Universal Robots PolyScope program: Main Program Left noweld.urp

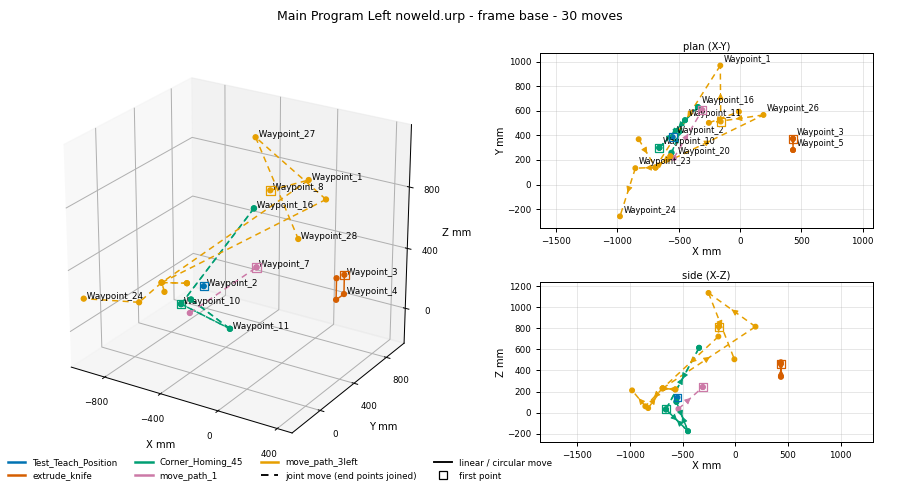
[picture p0: tool path of Main Program Left noweld.urp in frame base, 30 of 65 moves have a stored position in this frame; points joined in program order, loops and branches not executed]
Program Main Program Left noweld (installation=default directory=/programs createdIn=5.14.5 lastSavedIn=5.14.5 robotSerialNumber=20236801216)
Calibrated DH parameters: a=[-0.000021, -0.748897, -0.28186, -0.00004, -0.000055, 0]; d=[0.236225, -424.082933, -1564.66872, 1988.95162, 0.159094, 0.153873]; alpha=[1.570844, 0.001002, 0.000337, 1.571488, -1.569996, 0]; deltaTheta=[0, -0.516316, 5.626292, 1.173211, 0.000001, 0]
InitVariablesNode variables(variable(name=freedrive_m_var, expression=False))
Robot Program (runOnlyOnce=true)
  'start of main program'
  SafeHome (positionOptionType=SPEED_AND_ACCELERATION speed=1.047198 acceleration=1.396263 nextMotionTime=2)
  Set NoAction tcp=pretend_w_top
  Script: Test_Teach_Position()
  Set NoAction tcp=pretend_w_top
  Script: Corner_Homing_45()
  Set NoAction tcp=pretend_welder
  Script: extrude_knife()
  Script file /programs/analyze_touchpoints.script
    | # this file creates the function for analyzing touchpoints
    | # define pi
    | pi = 3.1415926535
    | 
    | # this is the main entry point for calculations.
    | # it takes in the 5 points, analyzes the shape of the box, and then calculates path points and returns them
    | # specifically for Down, Over, then Around (DOtA)
    | # specifically for right-sided boxes (vertical weld on right side of edge)
    | def main_calculate_right(p11, p12, p21, p22, p3, p13, p23):
    |     struct1 = analyze_touchpoints_only(p11, p12, p21, p22, p3)
    |     list1 = analyze_vertical_touchpoints(p11, p12, p13, p21, p22, p23, p3)
    |     struct2 = calculate_DOtA_points_right(struct1, list1)
    |     return struct2
    | end
    | 
    | # this is the main entry point for calculations.
    | # it takes in the 5 points, analyzes the shape of the box, and then calculates path points and returns them
    | # specifically for Down, Over, then Around (DOtA)
    | # specifically for left-sided boxes (vertical weld on left side of edge)
    | def main_calculate_left(p11, p12, p21, p22, p3):
    |     struct1 = analyze_touchpoints_only(p11, p12, p21, p22, p3)
    |     struct2 = calculate_DOtA_points_left(struct1)
    |     return struct2
    | end
    | 
    | # it takes 5 arguments as points
    | # it returns a struct containing: (pointintersect, pointapproach1, pointapproach2, point1, point2, point3, point4, point5, pointreturn1, heading1, heading2, heading3, path2r1, path2r2, path2l1, path2l2)
    | # specifically for Around then Up (AtU)
    | def analyze_touchpoints(p11, p12, p21, p22, p3):
    |   # FIND THE INTERSECTION
    |   # comment get the z
    |   zcoord=p3[2]
    | 
    |   # get the raw points from the first line
    |   l1p1x=p11[0]
    |   l1p1y=p11[1]
    |   l1p2x=p12[0]
    |   l1p2y=p12[1]
    | 
    |   # equate the first line in 2d space
    |   ml1 = (l1p2y-l1p1y) / (l1p2x-l1p1x)
    | 
    |   # b = y - mx
    |   bl1 = l1p1y - ml1 * l1p1x
    | 
    |   # get the raw points from the second line
    |   l2p1x=p21[0]
    |   l2p1y=p21[1]
    |   l2p2x=p22[0]
    |   l2p2y=p22[1]
    | 
    |   # equate the second line in 2d space
    |   ml2 = (l2p2y-l2p1y) / (l2p2x-l2p1x)
    | 
    |   # b = y - mx
    |   bl2 = l2p1y - ml2 * l2p1x
    | 
    | 
    |   # find the intersection of the two lines
    |   # m1x+b1 = m2x+b2
    |   # m1x - m2x = b2 - b1
    |   # x = (b2-b1) / (m1-m2)
    |   xintersect = (bl2-bl1) / (ml1-ml2)
    |   yintersect = ml1 * xintersect + bl1
    | 
    |   #FIND THE VECTORS
    |   #define a vector from the intersection to the second point on the first line
    |   l1delxfull = l1p2x - xintersect
    |   l1delyfull = l1p2y - yintersect
    | 
    |   l1delmag = sqrt(l1delxfull*l1delxfull + l1delyfull*l1delyfull)
    | 
    |   l1delxunit = l1delxfull / l1delmag
    |   l1delyunit = l1delyfull / l1delmag
    | 
    |   #define a vector from the intersection to the second point on the second line
    |   l2delxfull = l2p2x - xintersect
    |   l2delyfull = l2p2y - yintersect
    | 
    |   l2delmag = sqrt(l2delxfull*l2delxfull + l2delyfull*l2delyfull)
    | 
    |   l2delxunit = l2delxfull / l2delmag
    |   l2delyunit = l2delyfull / l2delmag
    | 
    |   # FIND THE FOUR POINTS ON THE LINES
    |   # find locations 8 inches away from  intersect point
    |   # CONST
    |   welddistance = 8
    |   roundoverdistance = 0.05
    |   zup = .375
    |   # inches
    |   wd = welddistance * 25.4 / 1000
    |   rod = roundoverdistance * 25.4 / 1000
    |   zup = zup * 25.4 / 1000
    | 
    |   # now we have the unit vector. extend the weld distance from the intersection
    |   x = xintersect + l1delxunit * wd
    |   y = yintersect + l1delyunit * wd
    |   z = zcoord + zup
    | 
    |   point1 = p[x,y,z,1.570796,0,0] # dummy orientation for now
    | 
    |   x = xintersect + l1delxunit * rod
    |   y = yintersect + l1delyunit * rod
    | 
    |   point2 = p[x,y,z,1.570796,0,0]
    | 
    |   # now we have the unit vector. extend the weld distance from the intersection
    |   x = xintersect + l2delxunit * wd
    |   y = yintersect + l2delyunit * wd
    | 
    |   point5 = p[x,y,z,0,-1.570796,0]
    | 
    |   x = xintersect + l2delxunit * rod
    |   y = yintersect + l2delyunit * rod
    | 
    |   point4 = p[x,y,z,0,-1.570796,0]
    | 
    |   #DEFINE APPROACH POINTS
    |   pointintersect = p[xintersect,yintersect,zcoord,0,0,0]
    |   pointapproach1 = p[xintersect+0.1,yintersect+0.1,z,1.570796,0,0]
    |   pointapproach2 = p[point1[0], point1[1]+0.1, point1[2], point1[3], point1[4], point1[5]]
    |   pointreturn1 = p[point5[0]+0.1, point5[1], point5[2], point5[3], point5[4], point5[5]]
    | 
    |   #FIND HEADINGS
    |   #for each heading, find the angle of the line with respect to the pos x axis. then add/subtract 90 degrees because you want to be perpendicular to that
    |   headingvector1 = convert_uv_to_heading(l1delxunit, l1delyunit)
    |   headingvector2 = convert_uv_to_heading(l2delxunit, l2delyunit)
    |   # find halfway heading
    |   heading2 = (headingvector1 + headingvector2)/2
    |   # find headings that the robot should face while traveling, perpendicular to the vectors of the sides of the box
    |   heading1 = headingvector1 + pi/2
    |   heading3 = headingvector2 - pi/2
    | 
    |   #FIND POINT 3
    |   #see if we have to / can find point 3
    |   findpoint3 = True
    |   if roundoverdistance == 0:
    |     findpoint3 = False
    |   end
    |   if findpoint3:
    |     # i need to find the point3 such that the arc from p2 to p3 to p4 is tangent to p1-p2 and p4-p5. making this a smooth path will be good
    |     # the direction of movement is from pointintersect in the direction of heading2
    |     # how much movement though? this will depend on whether it is actually a 90 degree angle or not.
    |     # first, find the perpendicular lines through points 2 and 4
    |     perp2 = find_perpendicular_line(ml1, point2[0], point2[1])
    |     perp4 = find_perpendicular_line(ml2, point4[0], point4[1])
    |     # next, find the intersection of those two lines
    |     perpintersect = find_intersection(perp2[0], perp2[1], perp4[0], perp4[1])
    |     radiusofcircle = distance_between(perpintersect[0], perpintersect[1], 0, point2[0], point2[1], 0)
    |     # find a vector the direction of heading2
    |     uvx = cos(heading2)
    |     uvy = sin(heading2)
    |     # compute point3. pass in negative radius because the direction is into the tank but we want to move from the intersection out to the rounded edge.
    |     point3coords = add_vectordistance_to_point(perpintersect[0], perpintersect[1], z, uvx, uvy, 0, -1 * radiusofcircle)
    |     point3 = p[point3coords[0], point3coords[1], point3coords[2], 0, 0, 0]
    |   end
    | 
    |   #APPLY ACTUAL RXRYRZ TO POINTS
    |   # convert the headings to rxryrz and insert those values into the relevant points
    |   rxryrz = convert_heading_to_axang(heading1)
    |   rx = rxryrz[0]
    |   ry = rxryrz[1]
    |   rz = rxryrz[2]
    |   pointapproach1 = p[pointapproach1[0], pointapproach1[1], pointapproach1[2], rx, ry, rz]
    |   pointapproach2 = p[pointapproach2[0], pointapproach2[1], pointapproach2[2], rx, ry, rz]
    |   point1 = p[point1[0], point1[1], point1[2], rx, ry, rz]
    |   point2 = p[point2[0], point2[1], point2[2], rx, ry, rz]
    |   rxryrz = convert_heading_to_axang(heading2)
    |   rx = rxryrz[0]
    |   ry = rxryrz[1]
    |   rz = rxryrz[2]
    |   if findpoint3:
    |     point3 = p[point3[0], point3[1], point3[2], rx, ry, rz]
    |   else:
    |     point3 = point2
    |   end
    |   rxryrz = convert_heading_to_axang(heading3)
    |   rx = rxryrz[0]
    |   ry = rxryrz[1]
    |   rz = rxryrz[2]
    |   point4 = p[point4[0], point4[1], point4[2], rx, ry, rz]
    |   point5 = p[point5[0], point5[1], point5[2], rx, ry, rz]
    |   pointreturn1 = p[pointreturn1[0], pointreturn1[1], pointreturn1[2], rx, ry, rz]
    | 
    |   #find path2 (the part that goes up)
    |   four_vertical_points = find_vertical_points(pointintersect, l1delxunit, l1delyunit, l2delxunit, l2delyunit, zup, wd, heading1, heading3)
    |   path2r1 = four_vertical_points[0]
    |   path2r2 = four_vertical_points[1]
    |   path2l1 = four_vertical_points[2]
    |   path2l2 = four_vertical_points[3]
    | 
    |   #RETURN STRUCT
    |   ret = struct(pointintersect=pointintersect, pointapproach1=pointapproach1, pointapproach2=pointapproach2, point1=point1, point2=point2, point3=point3, point4=point4, point5=point5, pointreturn1=pointreturn1, heading1=heading1, heading2=heading2, heading3=heading3, path2r1=path2r1, path2r2=path2r2, path2l1=path2l1, path2l2=path2l2)
    |   return ret
    | end
    | 
    | # it takes 5 arguments as points
    | # it returns a struct containing: (pointintersect, heading1, heading2, heading3, l1delxunit, l1delyunit, l2delxunit, l2delyunit)
    | def analyze_touchpoints_only(p11, p12, p21, p22, p3):
    |   # FIND THE INTERSECTION
    |   # comment get the z
    |   zcoord=p3[2]
    | 
    |   # get the raw points from the first line
    |   l1p1x=p11[0]
    |   l1p1y=p11[1]
    |   l1p2x=p12[0]
    |   l1p2y=p12[1]
    | 
    |   # equate the first line in 2d space
    |   ml1 = (l1p2y-l1p1y) / (l1p2x-l1p1x)
    | 
    |   # b = y - mx
    |   bl1 = l1p1y - ml1 * l1p1x
    | 
    |   # get the raw points from the second line
    |   l2p1x=p21[0]
    |   l2p1y=p21[1]
    |   l2p2x=p22[0]
    |   l2p2y=p22[1]
    | 
    |   # equate the second line in 2d space
    |   ml2 = (l2p2y-l2p1y) / (l2p2x-l2p1x)
    | 
    |   # b = y - mx
    |   bl2 = l2p1y - ml2 * l2p1x
    | 
    | 
    |   # find the intersection of the two lines
    |   # m1x+b1 = m2x+b2
    |   # m1x - m2x = b2 - b1
    |   # x = (b2-b1) / (m1-m2)
    |   xintersect = (bl2-bl1) / (ml1-ml2)
    |   yintersect = ml1 * xintersect + bl1
    | 
    |   pointintersect = p[xintersect,yintersect,zcoord,0,0,0]
    | 
    |   #FIND THE VECTORS
    |   #define a vector from the intersection to the second point on the first line
    |   l1delxfull = l1p2x - xintersect
    |   l1delyfull = l1p2y - yintersect
    | 
    |   l1delmag = sqrt(l1delxfull*l1delxfull + l1delyfull*l1delyfull)
    | 
    |   l1delxunit = l1delxfull / l1delmag
    |   l1delyunit = l1delyfull / l1delmag
    | 
    |   #define a vector from the intersection to the second point on the second line
    |   l2delxfull = l2p2x - xintersect
    |   l2delyfull = l2p2y - yintersect
    | 
    |   l2delmag = sqrt(l2delxfull*l2delxfull + l2delyfull*l2delyfull)
    | 
    |   l2delxunit = l2delxfull / l2delmag
    |   l2delyunit = l2delyfull / l2delmag
    | 
    |   #FIND HEADINGS
    |   #for each heading, find the angle of the line with respect to the pos x axis. then add/subtract 90 degrees because you want to be perpendicular to that
    |   headingvector1 = convert_uv_to_heading(l1delxunit, l1delyunit)
    |   headingvector2 = convert_uv_to_heading(l2delxunit, l2delyunit)
    |   # find halfway heading
    |   heading2 = (headingvector1 + headingvector2)/2
    |   # find headings that the robot should face while traveling, perpendicular to the vectors of the sides of the box
    |   heading1 = headingvector1 + pi/2
    |   heading3 = headingvector2 - pi/2
    | 
    |   #RETURN STRUCT
    |   ret = struct(pointintersect=pointintersect, heading1=heading1, heading2=heading2, heading3=heading3, l1delxunit=l1delxunit, l1delyunit=l1delyunit, l2delxunit=l2delxunit, l2delyunit=l2delyunit)
    |   return ret
    | end
    | 
    | # given a struct from analyze_touchpoints_only(), calculate the points
    | def calculate_DOtA_points_right(struct1, listleans):
    |     # get the stuff from the struct
    |     pointintersect = struct1[0]
    |     heading1 = struct1[1]
    |     heading2 = struct1[2]
    |     heading3 = struct1[3]
    |     l1delxunit = struct1[4]
    |     l1delyunit = struct1[5]
    |     l2delxunit = struct1[6]
    |     l2delyunit = struct1[7]
    | 
    |     # FIND THE POINTS ON THE LINES OF THE FIRST TURN PATH
    |     # find locations 8 inches away from  intersect point
    |     # CONST
    |     welddistance1 = 8 # vertical weld distance
    |     welddistance2 = 6 # first path second leg
    |     welddistance3 = 8 # second path second leg
    |     zup = .375
    |     # inches
    |     wd1 = welddistance1 * 25.4 / 1000
    |     wd2 = welddistance2 * 25.4 / 1000
    |     wd3 = welddistance3 * 25.4 / 1000
    |     zup = zup * 25.4 / 1000
    | 
    |     x = pointintersect[0] + l1delxunit * zup
    |     y = pointintersect[1] + l1delyunit * zup
    |     z = pointintersect[2] + zup
    | 
    |     #apply actual rxryrz to points
    |     # convert the headings to rxryrz and insert those values into the relevant points
    |     rxryrz = convert_heading_to_axang_preheatdown(heading1)
    |     rx = rxryrz[0]
    |     ry = rxryrz[1]
    |     rz = rxryrz[2]
    | 
    |     point1 = p[x + wd1*listleans[0], y + wd1*listleans[1], z + wd1, rx, ry, rz] # add in the listleans factor to follow the face of the box as we move up
    |     point2 = p[x, y, z, rx, ry, rz]
    | 
    |     # convert the headings to rxryrz and insert those values into the relevant points
    |     rxryrz = convert_heading_to_axang_ccw(heading1)
    |     rx = rxryrz[0]
    |     ry = rxryrz[1]
    |     rz = rxryrz[2]
    | 
    |     point4 = p[x, y, z, rx, ry, rz]
    |     x = x + l1delxunit * wd2
    |     y = y + l1delyunit * wd2
    |     point5 = p[x, y, z, rx, ry, rz]
    | 
    |     # FIND THE POINTS ON THE LINES OF THE SECOND AROUND PATH
    |     roundoverdistance = 0.05
    |     rod = roundoverdistance * 25.4 / 1000
    | 
    |     # now we have the unit vector. extend the weld distance from the intersection
    |     x = pointintersect[0] + l1delxunit * (zup)
    |     y = pointintersect[1] + l1delyunit * zup
    |     # convert the headings to rxryrz and insert those values into the relevant points
    |     rxryrz = convert_heading_to_axang(heading1)
    |     rx = rxryrz[0]
    |     ry = rxryrz[1]
    |     rz = rxryrz[2]
    |     point_1 = p[x, y, z, rx, ry, rz]
    | 
    |     x = pointintersect[0] + l1delxunit * rod
    |     y = pointintersect[1] + l1delyunit * rod
    |     point_2 = p[x, y, z, rx, ry, rz]
    | 
    |     # now we have the unit vector. extend the weld distance from the intersection
    |     x = pointintersect[0] + l2delxunit * wd3
    |     y = pointintersect[1] + l2delyunit * wd3
    |     # convert the headings to rxryrz and insert those values into the relevant points
    |     rxryrz = convert_heading_to_axang(heading3)
    |     rx = rxryrz[0]
    |     ry = rxryrz[1]
    |     rz = rxryrz[2]
    |     point_5 = p[x, y, z, rx, ry, rz]
    | 
    |     x = pointintersect[0] + l2delxunit * rod
    |     y = pointintersect[1] + l2delyunit * rod
    |     point_4 = p[x, y, z, rx, ry, rz]
    | 
    |     #FIND POINT 3
    |     # by calling analyze_touchpoints()
    |     atret = analyze_touchpoints(point_2, point_1, point_4, point_5, pointintersect)
    |     point_3 = atret[5]
    | 
    | 
    |     struct2 = struct(point1=point1, point2=point2, point4=point4, point5=point5, point_1=point_1, point_2=point_2, point_3=point_3, point_4=point_4, point_5=point_5)
    |     return struct2
    | end
    | 
    | # given a struct from analyze_touchpoints_only(), calculate the points
    | def calculate_DOtA_points_left(struct1):
    |     # get the stuff from the struct
    |     pointintersect = struct1[0]
    |     heading1 = struct1[1]
    |     heading2 = struct1[2]
    |     heading3 = struct1[3]
    |     l1delxunit = struct1[4]
    |     l1delyunit = struct1[5]
    |     l2delxunit = struct1[6]
    |     l2delyunit = struct1[7]
    | 
    |     # FIND THE POINTS ON THE LINES OF THE FIRST TURN PATH
    |     # find locations 8 inches away from  intersect point
    |     # CONST
    |     welddistance = 8
    |     zup = .375
    |     # inches
    |     wd = welddistance * 25.4 / 1000
    |     zup = zup * 25.4 / 1000
    | 
    |     x = pointintersect[0] + l2delxunit * zup
    |     y = pointintersect[1] + l2delyunit * zup
    |     z = pointintersect[2] + zup
    | 
    |     #apply actual rxryrz to points
    |     # convert the headings to rxryrz and insert those values into the relevant points
    |     rxryrz = convert_heading_to_axang_preheatdown(heading3)
    |     rx = rxryrz[0]
    |     ry = rxryrz[1]
    |     rz = rxryrz[2]
    | 
    |     point1 = p[x, y, z + wd, rx, ry, rz]
    |     point2 = p[x, y, z, rx, ry, rz]
    | 
    |     # convert the headings to rxryrz and insert those values into the relevant points
    |     rxryrz = convert_heading_to_axang(heading3)
    |     rx = rxryrz[0]
    |     ry = rxryrz[1]
    |     rz = rxryrz[2]
    | 
    |     point4 = p[x, y, z, rx, ry, rz]
    |     x = x + l2delxunit * wd
    |     y = y + l2delyunit * wd
    |     point5 = p[x, y, z, rx, ry, rz]
    | 
    |     # FIND THE POINTS ON THE LINES OF THE SECOND AROUND PATH
    |     roundoverdistance = 0.05
    |     rod = roundoverdistance * 25.4 / 1000
    | 
    |     # now we have the unit vector. extend the weld distance from the intersection
    |     x = pointintersect[0] + l2delxunit * (zup)
    |     y = pointintersect[1] + l2delyunit * zup
    |     # convert the headings to rxryrz and insert those values into the relevant points
    |     rxryrz = convert_heading_to_axang_ccw(heading3)
    |     rx = rxryrz[0]
    |     ry = rxryrz[1]
    |     rz = rxryrz[2]
    |     point_1 = p[x, y, z, rx, ry, rz]
    | 
    |     x = pointintersect[0] + l2delxunit * rod
    |     y = pointintersect[1] + l2delyunit * rod
    |     point_2 = p[x, y, z, rx, ry, rz]
    | 
    |     # now we have the unit vector. extend the weld distance from the intersection
    |     x = pointintersect[0] + l1delxunit * wd
    |     y = pointintersect[1] + l1delyunit * wd
    |     # convert the headings to rxryrz and insert those values into the relevant points
    |     rxryrz = convert_heading_to_axang_ccw(heading1)
    |     rx = rxryrz[0]
    |     ry = rxryrz[1]
    |     rz = rxryrz[2]
    |     point_5 = p[x, y, z, rx, ry, rz]
    | 
    |     x = pointintersect[0] + l1delxunit * rod
    |     y = pointintersect[1] + l1delyunit * rod
    |     point_4 = p[x, y, z, rx, ry, rz]
    | 
    |     #FIND POINT 3
    |     # by calling analyze_touchpoints()
    |     atret = analyze_touchpoints(point_2, point_1, point_4, point_5, pointintersect)
    |     point_3 = atret[5]
    |     #point 3 will not have the correct rxryrz though because now the gun needs to be face up.
    |     rxryrz = convert_heading_to_axang_ccw(heading2)
    |     rx = rxryrz[0]
    |     ry = rxryrz[1]
    |     rz = rxryrz[2]
    |     point_3 = p[point_3[0], point_3[1], point_3[2], rx, ry, rz]
    | 
    |     struct2 = struct(point1=point1, point2=point2, point4=point4, point5=point5, point_1=point_1, point_2=point_2, point_3=point_3, point_4=point_4, point_5=point_5)
    |     return struct2
    | end
    | 
    | # this function analyzes the vertical points
    | # calculates the slope of the edge in question
    | # specifically, for each inch up in the z direction, what is the change in x and change in y direction
    | # returns a list of [nx, ny]
    | def analyze_vertical_touchpoints(p11, p12, p13, p21, p22, p23, p3):
    |     # first, find the equations of the planes from the 6 points
    |     plane1 = findplane(p11, p12, p13)
    |     plane2 = findplane(p21, p22, p23)
    |     # Find the Direction Vector of the Line: The direction vector d of the line of intersection can be found by taking the cross product of the normal vectors of each plane (a, b, and c)
    |     nx = plane1[1]*plane2[2] - plane1[2]*plane2[1]
    |     ny = plane1[2]*plane2[0] - plane1[0]*plane2[2]
    |     nz = plane1[0]*plane2[1] - plane1[1]*plane2[0]
    |     # normalize the vector so the z length is 1
    |     multiplier = 1 / nz
    |     nx = nx * multiplier
    |     ny = ny * multiplier
    |     nz = nz * multiplier # should become equal to 1
    |     ret = [nx, ny]
    |     return ret
    | end
    | 
    | # given 3 points, this finds the plane and its equation
    | # rereturns ax + by + cz + d = 0 in a list of [a, b, c, d]
    | def findplane(p11, p12, p13):
    |     # extract coordinates
    |     x1 = p11[0]
    |     y1 = p11[1]
    |     z1 = p11[2]
    |     x2 = p12[0]
    |     y2 = p12[1]
    |     z2 = p12[2]
    |     x3 = p13[0]
    |     y3 = p13[1]
    |     z3 = p13[2]
    |     # create vectors from the points
    |     v1x = x2-x1
    |     v1y = y2-y1
    |     v1z = z2-z1
    |     v2x = x3-x1
    |     v2y = y3-y1
    |     v2z = z3-z1
    |     #calculate the normal vector using the cross product
    |     nx = v1y*v2z - v1z*v2y # i component
    |     ny = v1z*v2x - v1x*v2z # j component
    |     nz = v1x*v2y - v1y*v2x # k component
    |     # calculate d in the plane equation
    |     d = -1 * (nx*x1 + ny*y1 + nz*z1)
    |     ret = [nx, ny, nz, d]
    |     return ret
    | end
    | 
    | # given a heading, (ccw from +x axis), find the mx+b slope
    | # fails if exactly vertical
    | def get_slope_from_heading(heading):
    |     return tan(heading)
    | end
    | 
    | 
    | 
    | # this function finds the points (and rxryrz) of the 2 points (start and end) of vertical weld section
    | def find_vertical_points(pointintersect, l1delxunit, l1delyunit, l2delxunit, l2delyunit, offset, wd, heading1, heading3):
    | 
    |   # find right side stuff
    |   # find the point in 3d space that is .375 up and .375 over
    |   x = pointintersect[0] + l1delxunit * offset
    |   y = pointintersect[1] + l1delyunit * offset
    |   z = pointintersect[2] + offset
    |   # find rxryrz
    |   rxryrz = convert_heading_to_axang_preheatup(heading1)
    |   rx = rxryrz[0]
    |   ry = rxryrz[1]
    |   rz = rxryrz[2]
    |   path2r1 = p[x, y, z, rx, ry, rz]
    |   path2r2 = p[x, y, z + wd, rx, ry, rz]
    | 
    |   # find left side
    |   # find the point in 3d space that is .375 up and .375 over
    |   x = pointintersect[0] + l2delxunit * offset
    |   y = pointintersect[1] + l2delyunit * offset
    |   z = pointintersect[2] + offset
    |   # find rxryrz
    |   rxryrz = convert_heading_to_axang_preheatup(heading3)
    |   rx = rxryrz[0]
    |   ry = rxryrz[1]
    |   rz = rxryrz[2]
    |   path2l1 = p[x, y, z, rx, ry, rz]
    |   path2l2 = p[x, y, z + wd, rx, ry, rz]
    | 
    |   ret = struct(path2r1=path2r1, path2r2=path2r2, path2l1=path2l1, path2l2=path2l2)
    |   return ret
    | end
    | 
    | # this function converts a unit vector to its heading angle ccw from x+ axis
    | # takes uvx and uvy
    | # returns heading in radians
    | def convert_uv_to_heading(uvx, uvy):
    |   baseang = atan(uvy/uvx)
    |   if uvx < 0:
    |     ang = baseang + pi
    |   elif uvy < 0:
    |     ang = baseang + pi * 2
    |   else:
    |     ang = baseang
    |   end
    |   return ang
    | end
    | 
    | # this function finds the equation of a line, perpendicular to a given line, and going through a given point
    | # takes 3 arguments: m (the original line's slope), x (point's x coord), y (point's y coord). the b of the original line is not needed
    | # returns a list of [m,b] (the slope and intercept of the new line)
    | def find_perpendicular_line(origm, x, y):
    |   m = (1/origm) * -1
    |   b = y - m*x
    |   ret = [m, b]
    |   return ret
    | end
    | 
    | # this function finds the intersection point between two lines in the xy plane
    | # takes 4 arguments: m1, b1, m2, b2
    | # returns a list of [x,y] (the point of intersection)
    | def find_intersection(m1, b1, m2, b2):
    |   # m1x+b1 = m2x+b2
    |   # m1x - m2x = b2 - b1
    |   # x = (b2-b1) / (m1-m2)
    |   x = (b2-b1) / (m1-m2)
    |   y = m1 * x + b1
    |   ret = [x, y]
    |   return ret
    | end
    | 
    | # this function finds the distance between 2 points in 3d space
    | # it takes 6 arguments: x1, y1, z1, x2, y2, z2
    | # it returns a distance
    | def distance_between(x1, y1, z1, x2, y2, z2):
    |   distsquared = (x2-x1)*(x2-x1)+(y2-y1)*(y2-y1)+(z2-z1)*(z2-z1)
    |   dist = sqrt(distsquared)
    |   return dist
    | end
    | 
    | # this function takes a point, a unit vector, and a distance, and adds the distance to the point in the direction of the unit vector (3d space)
    | # it returns a point as a list of coordinates
    | def add_vectordistance_to_point(xi, yi, zi, uvx, uvy, uvz, delta):
    |   xf = xi + uvx * delta
    |   yf = yi + uvy * delta
    |   zf = zi + uvz * delta
    |   ret = [xf, yf, zf]
    |   return ret
    | end
    | 
    | # this function converts a heading (ccw radians from the positive x axis) into rxryrz to be put into a point p[]
    | # this will point the gun in this heading with the bottom side of the gun facing up.
    | # the values used in this program were calculated by doing rotation matrix math in the file on WI-CALVINB10 C. Documents. Theory for converting rotations into axis angle representations
    | def convert_heading_to_axang(heading):
    |  axisxraw = -1 * sin(heading)
    |  axisyraw = cos(heading) + 1
    |  axiszraw = sin(heading)
    | 
    |  magnitude = sqrt(axisxraw*axisxraw + axisyraw*axisyraw + axiszraw*axiszraw)
    | 
    |  axisxunit = axisxraw / magnitude
    |  axisyunit = axisyraw / magnitude
    |  axiszunit = axiszraw / magnitude
    | 
    |  angle = acos( (cos(heading) - 1) / 2 )
    | 
    |  rxout = axisxunit * angle
    |  ryout = axisyunit * angle
    |  rzout = axiszunit * angle
    | 
    |  return [rxout, ryout, rzout]
    | end
    | 
    | # this function converts a heading (ccw radians from the positive x axis) into rxryrz to be put into a point p[]
    | # this will point the gun in this heading with the preheat side of the gun tip facing up. Used for welding in a vertical path.
    | # the values used in this program were calculated by doing rotation matrix math in the file on WI-CALVINB10 C. Documents. Theory for converting rotations into axis angle representations
    | def convert_heading_to_axang_preheatup(heading):
    |  axisxraw = -sin(heading) + 1
    |  axisyraw = cos(heading)
    |  axiszraw = cos(heading)
    | 
    |  magnitude = sqrt(axisxraw*axisxraw + axisyraw*axisyraw + axiszraw*axiszraw)
    | 
    |  axisxunit = axisxraw / magnitude
    |  axisyunit = axisyraw / magnitude
    |  axiszunit = axiszraw / magnitude
    | 
    |  angle = acos( (-sin(heading) - 1) / 2 )
    | 
    |  rxout = axisxunit * angle
    |  ryout = axisyunit * angle
    |  rzout = axiszunit * angle
    | 
    |  return [rxout, ryout, rzout]
    | end
    | 
    | # this function converts a heading (ccw radians from the positive x axis) into rxryrz to be put into a point p[]
    | # this will point the gun in this heading with the preheat side of the gun tip facing down. Used for welding in a vertical path downwards.
    | # the values used in this program were calculated by doing rotation matrix math in the file on WI-CALVINB10 C. Documents. Theory for converting rotations into axis angle representations
    | def convert_heading_to_axang_preheatdown(heading):
    |  axisxraw = -sin(heading) - 1
    |  axisyraw = cos(heading)
    |  axiszraw = -cos(heading)
    | 
    |  magnitude = sqrt(axisxraw*axisxraw + axisyraw*axisyraw + axiszraw*axiszraw)
    | 
    |  axisxunit = axisxraw / magnitude
    |  axisyunit = axisyraw / magnitude
    |  axiszunit = axiszraw / magnitude
    | 
    |  angle = acos( (sin(heading) - 1) / 2 )
    | 
    |  rxout = axisxunit * angle
    |  ryout = axisyunit * angle
    |  rzout = axiszunit * angle
    | 
    |  return [rxout, ryout, rzout]
    | end
    | 
    | # this function converts a heading (ccw radians from the positive x axis) into rxryrz to be put into a point p[]
    | # this will point the gun in this heading with the preheat side of the gun tip facing right. Used for welding counterclockwise around the box.
    | # the values used in this program were calculated by doing rotation matrix math in the file on WI-CALVINB10 C. Documents. Theory for converting rotations into axis angle representations
    | def convert_heading_to_axang_ccw(heading):
    |  axisxraw = -sin(heading)
    |  axisyraw = cos(heading) - 1
    |  axiszraw = -sin(heading)
    | 
    |  magnitude = sqrt(axisxraw*axisxraw + axisyraw*axisyraw + axiszraw*axiszraw)
    | 
    |  axisxunit = axisxraw / magnitude
    |  axisyunit = axisyraw / magnitude
    |  axiszunit = axiszraw / magnitude
    | 
    |  angle = acos( (-cos(heading) - 1) / 2 )
    | 
    |  rxout = axisxunit * angle
    |  ryout = axisyunit * angle
    |  rzout = axiszunit * angle
    | 
    |  return [rxout, ryout, rzout]
    | end
    | 
    | # this function is for getting the points along the path of the corner homing 45
    | # point0 is the point where they touched
    | def get_corner_homing_45_pathpoints(point0):
    |   p0x = point0[0]
    |   p0y = point0[1]
    |   p0z = point0[2]
    |   p0rx = point0[3]
    |   p0ry = point0[4]
    |   p0rz = point0[5]
    | 
    |   #constants
    |   #distances of how far away from point the touchpoints are
    |   d0 = 0.15 # how far from the box to retreat and approach
    |   d1 = 0.05 # first distance from init point
    |   d2 = 0.2 # second distance from init point
    |   d3 = 0.125 #vertical distance from first point
    |   sqrt2 = 0.707106781
    | 
    |   ph1 = p[p0x + d0, p0y, p0z + .05, p0rx, p0ry, p0rz] #approach point for turn
    | 
    |   ph2 = p[p0x+d0-d0*sqrt2-sqrt2*d1, p0y+d0*sqrt2+sqrt2*d1, p0z+.05, .445, -1.562, .483]
    |   ph3 = p[p0x+d0-d0*sqrt2-sqrt2*d2, p0y+d0*sqrt2+sqrt2*d2, p0z+.05, .445, -1.562, .483]
    |   ph4 = p[p0x+d0-d0*sqrt2-sqrt2*d1, p0y-d0*sqrt2-sqrt2*d1, p0z+.05, 1.699, 3.576, 1.841]
    |   ph5 = p[p0x+d0-d0*sqrt2-sqrt2*d2, p0y-d0*sqrt2-sqrt2*d2, p0z+.05, 1.699, 3.576, 1.841]
    | 
    |   # go back to ph1
    |   ph6 = p[p0x + .05, p0y, p0z -.05, 0, 0, 0] # approach point for under turn
    |   # moveL from ph1 to ph6
    |   ph7 = p[p0x-.05, p0y, p0z-.05, 0, 0, 0]
    | 
    |   # add the vertical touch points
    |   ph2up = p[ph2[0], ph2[1], ph2[2]+d3, ph2[3], ph2[4], ph2[5]]
    |   ph4up = p[ph4[0], ph4[1], ph4[2]+d3, ph4[3], ph4[4], ph4[5]]
    |   ret = struct(ph1=ph1, ph2=ph2, ph3=ph3, ph4=ph4, ph5=ph5, ph6=ph6, ph7=ph7, ph2up=ph2up, ph4up=ph4up)
    |   return ret
    | end
  SuppressedNode
    path1 := analyze_touchpoints(p11,p12,p21,p22,p3)
  SuppressedNode
    Call move_path_1
  SuppressedNode
    MoveJ speed 60 deg/s, acceleration 80 deg/s^2 (useActiveTCP=true) feature=Base
      Waypoint Waypoint_19: TCP in base x=-539.433 y=254.004 z=21.521 mm, rx=-1.7232 ry=0.9213 rz=1.7071 rad; joints [-41.97, -63.602, 146.502, 9.159, 84.533, 189.272] deg; TCP offset x=8.55 y=-271.52 z=102 mm, rx=1.2092 ry=-1.2092 rz=1.2092 rad
  pathturn := main_calculate_left(p11,p12,p21,p22,p3)
  SuppressedNode
    Popup Message (haltProgram=false inputType=Variable) variable=pathturn
  Call move_path_3left
  SafeHome (positionOptionType=SPEED_AND_ACCELERATION speed=1.047198 acceleration=1.396263 nextMotionTime=2)
SubProgram -> move_path_3left
SubProgram Test_Teach_Position (keepSynchronizedWithDisk=false) programFile=/programs/Test Teach Position.urp
  SafeHome (positionOptionType=SPEED_AND_ACCELERATION speed=1.047198 acceleration=1.396263 nextMotionTime=2)
  SuppressedNode
    MoveL speed 250 mm/s, acceleration 1200 mm/s^2 (useActiveTCP=true) feature=Base
      Waypoint Waypoint_1: TCP in base x=183.613 y=373.491 z=464.002 mm, rx=0 ry=3.1416 rz=0 rad; joints [-144.817, -120.486, 148.461, -117.931, -90.033, 125.101] deg; TCP offset x=0 y=0 z=19 mm, rx=0 ry=0 rz=0 rad
      'move welder up out of holder'
  MoveJ speed 60 deg/s, acceleration 80 deg/s^2 (useActiveTCP=false) tcp=TCP_1_plate; feature=Base
    Waypoint Waypoint_2: TCP in base x=-548.957 y=386.285 z=143.71 mm, rx=1.5708 ry=0 rz=0 rad; joints [-60.253, -57.926, 123.544, -65.529, -60.311, -0.099] deg
  freedrive_m_var := False
  freedrive_m_var := True
  Popup Message (haltProgram=false message=Move the robot to the peg center, then click 'Continue' inputType=Text)
  freedrive_m_var := False
  Wait Sleep waitTime=0.25
  Script: sync()
  tcp_pose := get_actual_joint_positions()
SuppressedNode
  SubProgram -> move_path_1
SubProgram extrude_knife (keepSynchronizedWithDisk=false) programFile=/programs/extrude_knife.urp
  'Move to bucket'
  MoveJ speed 60 deg/s, acceleration 80 deg/s^2 (useActiveTCP=true) feature=Base
    Waypoint Waypoint_3: TCP in base x=432.121 y=373.496 z=463.993 mm, rx=0 ry=-3.1416 rz=0 rad; joints [-159.589, -103.956, 140.658, -126.656, -90.019, 110.321] deg
  MoveL speed 250 mm/s, acceleration 1200 mm/s^2 (useActiveTCP=true) feature=Base
    Waypoint Waypoint_4: TCP in base x=432.138 y=373.502 z=340.884 mm, rx=0 ry=3.1416 rz=0 rad; joints [-159.596, -94.144, 147.137, -142.947, -90.01, 110.313] deg
  'extrude out a foot'
  Wait Sleep waitTime=6
  MoveL speed 40 mm/s, acceleration 1200 mm/s^2 (useActiveTCP=true) feature=Base
    'slice over knife'
    Waypoint Waypoint_5: TCP in base x=432.16 y=281.352 z=340.893 mm, rx=0 ry=3.1416 rz=0 rad; joints [-169.69, -98.838, 150.801, -141.919, -90.013, 100.22] deg
  MoveL speed 250 mm/s, acceleration 1200 mm/s^2 (useActiveTCP=true) feature=Base
    Waypoint Waypoint_6: TCP in base x=432.128 y=281.346 z=478.493 mm, rx=0 ry=-3.1416 rz=0 rad; joints [-169.679, -110.118, 142.836, -122.671, -90.025, 100.232] deg
    'raise up away from knife'
  SafeHome (positionOptionType=SPEED_AND_ACCELERATION speed=1.047198 acceleration=1.396263 nextMotionTime=2)
SubProgram align_tcp_left (keepSynchronizedWithDisk=false) programFile=/programs/align_tcp_left.urp
  'this program aligns the tcp parallel to the y direction'
  cp := get_actual_tcp_pose()
  aligned_y_pose := p[cp[0],cp[1],cp[2],1.570796,0,0]
  MoveJ speed 60 deg/s, acceleration 80 deg/s^2 (useActiveTCP=true) feature=Base
    Waypoint Variable (Variable): variable=aligned_y_pose
SubProgram align_tcp_forward (keepSynchronizedWithDisk=false) programFile=/programs/align_tcp_forward.urp
  'this program aligns the tcp parallel to the y direction'
  cp := get_actual_tcp_pose()
  aligned_y_pose := p[cp[0],cp[1],cp[2],0,-1.570796,0]
  MoveJ speed 60 deg/s, acceleration 80 deg/s^2 (useActiveTCP=true) feature=Base
    Waypoint Variable (Variable): variable=aligned_y_pose
SubProgram align_tcp_up (keepSynchronizedWithDisk=false) programFile=/programs/align_tcp_up.urp
  'this program aligns the tcp parallel to the y direction'
  cp := get_actual_tcp_pose()
  aligned_y_pose := p[cp[0],cp[1],cp[2],0,0,0]
  MoveJ speed 60 deg/s, acceleration 80 deg/s^2 (useActiveTCP=true) feature=Base
    Waypoint Variable (Variable): variable=aligned_y_pose
SubProgram Corner_Homing_45 (keepSynchronizedWithDisk=false) programFile=/programs/Corner Homing 45.urp
  'Use this program when tool is already positioned close to corner at 45deg'
  'tool flange will seek all 3 sides. will save those 5 locs in p__'
  Set NoAction tcp=pretend_w_top
  'dummy move below for debug'
  SuppressedNode
    SafeHome (positionOptionType=SPEED_AND_ACCELERATION speed=1.047198 acceleration=1.396263 nextMotionTime=2)
  SuppressedNode
    MoveJ speed 60 deg/s, acceleration 80 deg/s^2 (useActiveTCP=true) feature=Base
      Waypoint Waypoint_1: TCP in base x=-726.76 y=313.857 z=-3.219 mm, rx=-0.1302 ry=-1.6605 rz=-0.1403 rad; joints [-65.067, -50.619, 153.092, -93.35, 35.027, 81.724] deg; TCP offset x=0 y=0 z=246 mm, rx=0 ry=0 rz=0 rad
      Waypoint Waypoint_2: TCP in base x=-1013.668 y=283.774 z=13.404 mm, rx=-0.1302 ry=-1.6605 rz=-0.1403 rad; joints [-36.803, -53.188, 133.142, -74.065, 63.057, 86.565] deg
  Wait Sleep waitTime=1
  tp := get_actual_tcp_pose()
  Script file /programs/analyze_touchpoints.script
    | (same text as the earlier copy of this file)
  path_pre := get_corner_homing_45_pathpoints(tp)
  ph1 := path_pre[0]
  ph2 := path_pre[1]
  ph3 := path_pre[2]
  ph4 := path_pre[3]
  ph5 := path_pre[4]
  ph6 := path_pre[5]
  ph7 := path_pre[6]
  MoveJ speed 60 deg/s, acceleration 80 deg/s^2 (useActiveTCP=true) feature=Base
    Waypoint Variable (Variable): variable=ph1
    Waypoint Variable (Variable): variable=ph2
  MoveL speed 50 mm/s, acceleration 100 mm/s^2 (useActiveTCP=true) feature=Base
    MoveDirectionNode expression=[-1,-1.0,0.0]
      Until TOOL_CONTACT_DETECTION (allowActions=false retraction=0 decelerationAcceleration=3 decelerationAngularAcceleration=34.906585)
  p11 := get_actual_tcp_pose()
  MoveJ speed 60 deg/s, acceleration 80 deg/s^2 (useActiveTCP=true) feature=Base
    Waypoint Variable (Variable): variable=ph3
  MoveL speed 50 mm/s, acceleration 100 mm/s^2 (useActiveTCP=true) feature=Base
    MoveDirectionNode expression=[-1,-1.0,0.0]
      Until TOOL_CONTACT_DETECTION (allowActions=false retraction=0 decelerationAcceleration=3 decelerationAngularAcceleration=34.906585)
  p12 := get_actual_tcp_pose()
  MoveJ speed 60 deg/s, acceleration 80 deg/s^2 (useActiveTCP=true) feature=Base
    Waypoint Variable (Variable): variable=ph3
    Waypoint Waypoint_10: TCP in base x=-658.265 y=299.53 z=30.91 mm, rx=0.4268 ry=-1.6215 rz=0.4371 rad; joints [-77.363, -55.591, 142.792, -102.186, -19.322, 105.94] deg
  MoveJ speed 20 deg/s, acceleration 80 deg/s^2 (useActiveTCP=true) feature=Base
    Waypoint Waypoint_11: TCP in base x=-448.863 y=524.6 z=-175.967 mm, rx=2.4733 ry=-1.8744 rz=0.2053 rad; joints [-65.056, -57.525, 139.86, -164.756, -91.924, 99.291] deg
    SuppressedNode
      Waypoint Waypoint_5: TCP in base x=-542.919 y=212.782 z=86.75 mm, rx=-0.746 ry=-1.5701 rz=-0.8083 rad; joints [-15.32, -63.738, 160.053, -88.648, -229.235, 89.501] deg
    Waypoint Waypoint_12: TCP in base x=-559.13 y=259.234 z=102.446 mm, rx=-0.8226 ry=-1.4861 rz=-0.8815 rad; joints [-31.871, -61.56, 166.811, -101.777, -239.831, 87.599] deg; TCP offset x=-1.157 y=-95.604 z=257.595 mm, rx=0 ry=0 rz=0 rad
  MoveJ speed 60 deg/s, acceleration 80 deg/s^2 (useActiveTCP=true) feature=Base
    Waypoint Variable (Variable): variable=ph4
  MoveL speed 50 mm/s, acceleration 100 mm/s^2 (useActiveTCP=true) feature=Base
    MoveDirectionNode expression=[-1.0,1.0,0.0]
      Until TOOL_CONTACT_DETECTION (allowActions=false retraction=0 decelerationAcceleration=3 decelerationAngularAcceleration=34.906585)
  p21 := get_actual_tcp_pose()
  MoveJ speed 60 deg/s, acceleration 80 deg/s^2 (useActiveTCP=true) feature=Base
    Waypoint Variable (Variable): variable=ph5
  MoveL speed 50 mm/s, acceleration 100 mm/s^2 (useActiveTCP=true) feature=Base
    MoveDirectionNode expression=[-1.0,1.0,0.0]
      Until TOOL_CONTACT_DETECTION (allowActions=false retraction=0 decelerationAcceleration=3 decelerationAngularAcceleration=34.906585)
  p22 := get_actual_tcp_pose()
  MoveJ speed 60 deg/s, acceleration 80 deg/s^2 (useActiveTCP=true) feature=Base
    Waypoint Variable (Variable): variable=ph5
    Waypoint Variable (Variable): variable=ph4
    SuppressedNode
      Waypoint Waypoint_5: TCP in base x=-542.919 y=212.782 z=86.75 mm, rx=-0.746 ry=-1.5701 rz=-0.8083 rad; joints [-15.32, -63.738, 160.053, -88.648, -229.235, 89.501] deg; TCP offset x=0 y=0 z=246 mm, rx=0 ry=0 rz=0 rad
    Waypoint Waypoint_13: TCP in base x=-559.13 y=259.234 z=102.446 mm, rx=-0.8226 ry=-1.4861 rz=-0.8815 rad; joints [-31.871, -61.56, 166.811, -101.777, -239.831, 87.599] deg; TCP offset x=-1.157 y=-95.604 z=257.595 mm, rx=0 ry=0 rz=0 rad
    Waypoint Waypoint_14: TCP in base x=-448.863 y=524.6 z=-175.967 mm, rx=2.4733 ry=-1.8744 rz=0.2053 rad; joints [-65.056, -57.525, 139.86, -164.756, -91.924, 99.291] deg; TCP offset x=0 y=0 z=246 mm, rx=0 ry=0 rz=0 rad
    Waypoint Waypoint_15: TCP in base x=-658.265 y=299.53 z=30.91 mm, rx=0.4268 ry=-1.6215 rz=0.4371 rad; joints [-77.363, -55.591, 142.792, -102.186, -19.322, 105.94] deg
    Waypoint Waypoint_16: TCP in base x=-343.952 y=632.142 z=615.175 mm, rx=-0.0259 ry=-0.0088 rz=-0.5675 rad; joints [-77.363, -55.591, 142.791, -175.721, 90.298, 134.942] deg
    Waypoint Variable (Variable): variable=ph6
    Waypoint Variable (Variable): variable=ph7
  MoveL speed 50 mm/s, acceleration 100 mm/s^2 (useActiveTCP=true) feature=Base
    MoveDirectionNode (selectedDirection=ZPlus)
      Until TOOL_CONTACT_DETECTION (allowActions=false retraction=0 decelerationAcceleration=3 decelerationAngularAcceleration=34.906585)
  p3 := get_actual_tcp_pose()
  MoveJ speed 60 deg/s, acceleration 80 deg/s^2 (useActiveTCP=true) feature=Base
    Waypoint Variable (Variable): variable=ph7
    Waypoint Variable (Variable): variable=ph6
    Waypoint Waypoint_17: TCP in base x=-343.952 y=632.142 z=615.175 mm, rx=-0.0259 ry=-0.0088 rz=-0.5675 rad; joints [-77.363, -55.591, 142.791, -175.721, 90.298, 134.942] deg
    Waypoint Waypoint_18: TCP in base x=-658.265 y=299.53 z=30.91 mm, rx=0.4268 ry=-1.6215 rz=0.4371 rad; joints [-77.363, -55.591, 142.792, -102.186, -19.322, 105.94] deg
  SafeHome (positionOptionType=SPEED_AND_ACCELERATION speed=1.047198 acceleration=1.396263 nextMotionTime=2)
  ''
  ''
  ''
  ''
  ''
  ''
Thread Thread_1 (runOnlyOnce=false)
  Loop While (checkContinuously=false) expression=True
    If freedrive_m_var≟ True
      Script: freedrive_mode()
    Else 
      Script: end_freedrive_mode()
    Script: sync()
SubProgram move_path_1 (keepSynchronizedWithDisk=false) programFile=/programs/move_path_2.urp
  pa1 := path1[1]
  pa2 := path1[2]
  p1 := path1[3]
  p2 := path1[4]
  p3 := path1[5]
  p4 := path1[6]
  p5 := path1[7]
  pr1 := path1[8]
  pvr1 := path1[12]
  pvr2 := path1[13]
  MoveJ speed 60 deg/s, acceleration 80 deg/s^2 (useActiveTCP=true) feature=Base
    SuppressedNode
      Waypoint Waypoint_9: TCP in base x=-308.524 y=606.099 z=242.383 mm, rx=-0.1348 ry=-3.0618 rz=-0.0522 rad; joints [-82.604, -97.742, 135.138, 229.977, -86.039, -167.57] deg; TCP offset x=0 y=0 z=260 mm, rx=0 ry=0 rz=0 rad
    Waypoint Waypoint_7: TCP in base x=-308.522 y=606.103 z=242.387 mm, rx=1.3699 ry=1.0669 rz=-1.2572 rad; joints [-84.673, -56.548, 94.558, 52.545, 94.971, 14.541] deg; TCP offset x=8.55 y=-265.17 z=108.77 mm, rx=1.2092 ry=-1.2092 rz=1.2092 rad
  MoveJ speed 60 deg/s, acceleration 80 deg/s^2 (useActiveTCP=true) feature=Base
    Waypoint Variable (Variable): variable=pa1
  MoveL speed 200 mm/s, acceleration 1200 mm/s^2 (useActiveTCP=true) feature=Base
    Waypoint Variable (Variable): variable(name=pa2)
  MoveL speed 50 mm/s, acceleration 1200 mm/s^2 (useActiveTCP=true) feature=Base
    Waypoint Variable (Variable): variable=p1
  Wait Sleep waitTime=1
  MoveL speed 12 mm/s, acceleration 1200 mm/s^2 (useActiveTCP=true) feature=Base
    Waypoint Variable (Variable): variable=p2
  MoveP speed 0.5 mm/s, acceleration 500 mm/s^2 (blendRadius=0.001 useActiveTCP=true) feature=Base
    CircleMove (OrientationMode=FIXED)
      Waypoint Variable (Variable): variable=p3
      Waypoint Variable (Variable): variable=p4
  MoveL speed 12 mm/s, acceleration 1200 mm/s^2 (useActiveTCP=true) feature=Base
    Waypoint Variable (Variable): variable=p5
  MoveL speed 250 mm/s, acceleration 1200 mm/s^2 (useActiveTCP=true) feature=Base
    Waypoint Variable (Variable): variable(name=pr1)
  SuppressedNode
    MoveJ speed 60 deg/s, acceleration 80 deg/s^2 (useActiveTCP=true) feature=Base
      Waypoint Variable (Variable): variable=pa1
  SuppressedNode
    MoveJ speed 60 deg/s, acceleration 80 deg/s^2 (useActiveTCP=true) feature=Base
      Waypoint Waypoint_8: TCP in base x=-372.861 y=716.17 z=314.677 mm, rx=1.5708 ry=0 rz=0 rad; joints [-79.161, -60.426, 105.047, -44.564, -79.226, 359.93] deg; TCP offset x=0 y=0 z=19 mm, rx=0 ry=0 rz=0 rad
  MoveJ speed 60 deg/s, acceleration 80 deg/s^2 (useActiveTCP=true) feature=Base
    Waypoint Waypoint_20: TCP in base x=-540.148 y=215.935 z=34.628 mm, rx=-1.5058 ry=1.0576 rz=1.5735 rad; joints [-25.659, -64.433, 142.414, 9.313, 85.709, 219.637] deg; TCP offset x=8.55 y=-271.52 z=102 mm, rx=1.2092 ry=-1.2092 rz=1.2092 rad
    Waypoint Waypoint_21: TCP in base x=-308.526 y=606.104 z=242.377 mm, rx=-2.1337 ry=0.3494 rz=2.1309 rad; joints [-106.376, -74.131, 126.55, 42.483, 90.905, 87.286] deg
  MoveJ speed 60 deg/s, acceleration 80 deg/s^2 (useActiveTCP=true) feature=Base
    Waypoint Variable (Variable): variable(name=pvr1)
  MoveL speed 50 mm/s, acceleration 100 mm/s^2 (useActiveTCP=true) feature=Base
    Waypoint Variable (Variable): variable(name=pvr2)
SubProgram move_path_3left (keepSynchronizedWithDisk=false) programFile=/programs/move_path_3left.urp
  'this is the path for Down, Over, then Back Around'
  ''
  SafeHome (positionOptionType=SPEED_AND_ACCELERATION speed=1.047198 acceleration=1.396263 nextMotionTime=2)
  MoveJ speed 60 deg/s, acceleration 80 deg/s^2 (useActiveTCP=true) feature=Base
    Waypoint Waypoint_8: TCP in base x=-157.621 y=513.354 z=815.678 mm, rx=-0.6727 ry=-1.8523 rz=-0.0554 rad; joints [-158.735, -104.322, 132.157, 58.275, -61.692, -46.244] deg; TCP offset x=-5.053 y=-331.71 z=103.574 mm, rx=1.2092 ry=-1.2092 rz=1.2092 rad
    Waypoint Waypoint_1: TCP in base x=-161.037 y=970.524 z=722.042 mm, rx=-0.555 ry=0.1065 rz=0.3286 rad; joints [-74.895, -76.586, 126.53, 213.07, -169.134, 52.325] deg; TCP offset x=-4.211 y=-279.829 z=105.916 mm, rx=1.2092 ry=-1.2092 rz=1.2092 rad
    Waypoint Waypoint_7: TCP in base x=-689.651 y=138.963 z=230.691 mm, rx=-0.852 ry=-1.646 rz=1.646 rad; joints [-53.938, -86.03, 160.535, 285.425, -269.23, 90.049] deg
    Waypoint Waypoint_9: TCP in base x=-568.725 y=230.602 z=220.208 mm, rx=-1.5191 ry=-0.5352 rz=0.574 rad; joints [-2.798, -73.075, 141.93, 288.829, -133.322, 87.786] deg; TCP offset x=8.385 y=-333.249 z=78.524 mm, rx=1.2092 ry=-1.2092 rz=1.2092 rad
    SuppressedNode
      Waypoint Waypoint_1: TCP in base x=-1177.596 y=138.956 z=230.69 mm, rx=-0.852 ry=-1.646 rz=1.646 rad; joints [-20.637, -63.427, 120.718, 302.664, -235.94, 90.036] deg; TCP offset x=-4.211 y=-279.829 z=105.916 mm, rx=1.2092 ry=-1.2092 rz=1.2092 rad
    SuppressedNode
      Waypoint Waypoint_2: TCP in base x=-689.651 y=138.963 z=230.691 mm, rx=-0.852 ry=-1.646 rz=1.646 rad; joints [-53.938, -86.03, 160.535, 285.425, -269.23, 90.049] deg
    SuppressedNode
      Waypoint Waypoint_3: TCP in base x=-161.037 y=970.524 z=722.042 mm, rx=-0.555 ry=0.1065 rz=0.3286 rad; joints [-74.895, -76.586, 126.53, 213.07, -169.134, 52.325] deg
    SuppressedNode
      SafeHome (positionOptionType=SPEED_AND_ACCELERATION speed=1.047198 acceleration=1.396263 nextMotionTime=2)
  ''
  p1 := pathturn[0]
  p2 := pathturn[1]
  p4 := pathturn[2]
  p5 := pathturn[3]
  MoveJ speed 60 deg/s, acceleration 80 deg/s^2 (useActiveTCP=true) feature=Base
    Waypoint Variable (Variable): variable=p1
  Wait Sleep waitTime=1
  MoveL speed 50 mm/s, acceleration 100 mm/s^2 (useActiveTCP=true) feature=Base
    Waypoint Variable (Variable): variable=p2
  Wait Sleep waitTime=1
  MoveL speed 20 mm/s, acceleration 5 mm/s^2 (useActiveTCP=true) feature=Base
    Waypoint Variable (Variable): variable=p4
  MoveL speed 50 mm/s, acceleration 100 mm/s^2 (useActiveTCP=true) feature=Base
    Waypoint Variable (Variable): variable=p5
  ''
  pret1 := p[p5[0]+.1,p5[1],p5[2],p5[3],p5[4],p5[5]]
  p_1 := pathturn[4]
  p_2 := pathturn[5]
  p_3 := pathturn[6]
  p_4 := pathturn[7]
  p_5 := pathturn[8]
  MoveJ speed 20 deg/s, acceleration 80 deg/s^2 (useActiveTCP=true) feature=Base
    Waypoint Variable (Variable): variable=pret1
    Waypoint Waypoint_22: TCP in base x=-568.725 y=230.602 z=220.208 mm, rx=-1.5191 ry=-0.5352 rz=0.574 rad; joints [-2.798, -73.075, 141.93, 288.829, -133.322, 87.786] deg; TCP offset x=8.385 y=-333.249 z=78.524 mm, rx=1.2092 ry=-1.2092 rz=1.2092 rad
    'now go into the ccw weld position'
    Waypoint Waypoint_7: TCP in base x=-689.651 y=138.963 z=230.691 mm, rx=-0.852 ry=-1.646 rz=1.646 rad; joints [-53.938, -86.03, 160.535, 285.425, -269.23, 90.049] deg; TCP offset x=-4.211 y=-279.829 z=105.916 mm, rx=1.2092 ry=-1.2092 rz=1.2092 rad
    ''
    Waypoint Waypoint_23: TCP in base x=-853.851 y=133.267 z=60.418 mm, rx=-0.2742 ry=-2.3597 rz=0.0468 rad; joints [-34.868, -57.997, 159.687, 213.62, -283.084, 21.643] deg; TCP offset x=8.385 y=-333.249 z=78.524 mm, rx=1.2092 ry=-1.2092 rz=1.2092 rad
    Waypoint Waypoint_24: TCP in base x=-979.398 y=-259.625 z=211.289 mm, rx=-0.673 ry=-1.4594 rz=-0.6402 rad; joints [21.182, -32.844, 122.516, 179.072, -269.511, -69.331] deg
    SuppressedNode
      Waypoint Waypoint_9: TCP in base x=-161.037 y=970.524 z=722.042 mm, rx=-0.555 ry=0.1065 rz=0.3286 rad; joints [-74.895, -76.586, 126.53, 213.07, -169.134, 52.325] deg; TCP offset x=-4.211 y=-279.829 z=105.916 mm, rx=1.2092 ry=-1.2092 rz=1.2092 rad
    SuppressedNode
      Waypoint Waypoint_22: TCP in base x=-308.534 y=606.085 z=242.393 mm, rx=1.3699 ry=1.0669 rz=-1.2572 rad; joints [-84.142, -55.374, 92.791, 53.186, 94.965, 15.074] deg
  SuppressedNode
    MoveP speed 20 mm/s, acceleration 2 mm/s^2 (blendRadius=0.001 useActiveTCP=true) feature=Base
      'below (until next comment) are points for testing out ccw circle weld'
      Waypoint Waypoint_8: TCP in base x=-1291.697 y=90.422 z=23.176 mm, rx=-0.673 ry=-1.4594 rz=-0.6402 rad; joints [-2.307, -18.609, 101.914, 185.717, -269.053, -45.852] deg; TCP offset x=8.385 y=-333.249 z=78.524 mm, rx=1.2092 ry=-1.2092 rz=1.2092 rad
      Waypoint Waypoint_10: TCP in base x=-1193.179 y=196.591 z=23.164 mm, rx=-0.673 ry=-1.4594 rz=-0.6402 rad; joints [-8.888, -18.95, 110.853, 177.226, -268.954, -39.273] deg
      Waypoint Waypoint_11: TCP in base x=-1193.173 y=196.572 z=23.158 mm, rx=0.078 ry=-1.5698 rz=0.1134 rad; joints [-28.391, -18.785, 116.78, 172.699, -268.884, 35.453] deg
      'end test points'
  MoveJ speed 60 deg/s, acceleration 80 deg/s^2 (useActiveTCP=true) feature=Base
    Waypoint Variable (Variable): variable=p_1
  MoveL speed 12 mm/s, acceleration 1200 mm/s^2 (useActiveTCP=true) feature=Base
    Waypoint Variable (Variable): variable=p_2
  MoveP speed 0.5 mm/s, acceleration 10 mm/s^2 (blendRadius=0.001 useActiveTCP=true) feature=Base
    CircleMove (OrientationMode=FIXED)
      Waypoint Variable (Variable): variable=p_3
      Waypoint Variable (Variable): variable=p_4
  MoveL speed 12 mm/s, acceleration 1200 mm/s^2 (useActiveTCP=true) feature=Base
    Waypoint Variable (Variable): variable=p_5
  SuppressedNode
    MoveL speed 250 mm/s, acceleration 1200 mm/s^2 (useActiveTCP=true) feature=Base
      Waypoint Waypoint_23: TCP in base x=-540.167 y=215.949 z=34.631 mm, rx=-1.5058 ry=1.0576 rz=1.5735 rad; joints [-26.452, -65.119, 143.749, 8.723, 85.674, 218.843] deg; TCP offset x=-4.211 y=-279.829 z=105.916 mm, rx=1.2092 ry=-1.2092 rz=1.2092 rad
  SuppressedNode
    MoveJ speed 60 deg/s, acceleration 80 deg/s^2 (useActiveTCP=true) feature=Base
      Waypoint Waypoint_24: TCP in base x=-308.526 y=606.096 z=242.373 mm, rx=-2.1337 ry=0.3494 rz=2.1309 rad; joints [-107.196, -73.784, 125.643, 43.029, 90.975, 86.468] deg
  MoveJ speed 60 deg/s, acceleration 80 deg/s^2 (useActiveTCP=true) feature=Base
    Waypoint Waypoint_25: TCP in base x=-826.866 y=369.358 z=43.114 mm, rx=0.575 ry=-1.4922 rz=0.5971 rad; joints [-59.333, -19.441, 121.825, 168.37, -269.932, 102.332] deg; TCP offset x=8.385 y=-333.249 z=78.524 mm, rx=1.2092 ry=-1.2092 rz=1.2092 rad
    Waypoint Waypoint_7: TCP in base x=-689.651 y=138.963 z=230.691 mm, rx=-0.852 ry=-1.646 rz=1.646 rad; joints [-53.938, -86.03, 160.535, 285.425, -269.23, 90.049] deg; TCP offset x=-4.211 y=-279.829 z=105.916 mm, rx=1.2092 ry=-1.2092 rz=1.2092 rad
  ''
  MoveJ speed 60 deg/s, acceleration 80 deg/s^2 (useActiveTCP=true) feature=Base
    Waypoint Waypoint_26: TCP in base x=191.113 y=567.512 z=815.514 mm, rx=-0.1358 ry=0.3961 rz=0.2088 rad; joints [-94.746, -100.957, 150.262, 188.452, -152.118, 48.82] deg; TCP offset x=-5.053 y=-331.71 z=103.574 mm, rx=1.2092 ry=-1.2092 rz=1.2092 rad
    Waypoint Waypoint_27: TCP in base x=-254.566 y=502.963 z=1135.402 mm, rx=-0.2619 ry=-0.7497 rz=1.349 rad; joints [-116.61, -108.45, 141.427, 125.702, -66.866, -29.172] deg
    Waypoint Waypoint_28: TCP in base x=-9.208 y=593.718 z=505.81 mm, rx=-1.4244 ry=-2.3441 rz=-0.5276 rad; joints [-167.145, -114.278, 136.39, 39.71, -32.494, -66.269] deg
    SuppressedNode
      Waypoint Waypoint_14: TCP in base x=436.687 y=409.759 z=815.514 mm, rx=-0.0352 ry=0.4178 rz=-0.2764 rad; joints [-122.957, -100.957, 150.262, 188.453, -152.119, 48.82] deg
    SuppressedNode
      Waypoint Waypoint_15: TCP in base x=412.386 y=384.342 z=1135.401 mm, rx=-0.6084 ry=-0.4075 rz=0.1224 rad; joints [-190.47, -108.449, 141.427, 125.702, -66.867, -29.172] deg
  ''
  ''
  ''
  ''
  ''
  ''
  SafeHome (positionOptionType=SPEED_AND_ACCELERATION speed=1.047198 acceleration=1.396263 nextMotionTime=2)
